TYPE (* logiBUS DI Events Struct Octal *)
  (* Version 1.0, 2026-05-28, franz *)
  PACKAGE logiBUS::io::DI;
  logiBUS_DI_Events_S_Octal : STRUCT
    Port1 : logiBUS::io::DI::logiBUS_DI_Events_S;
    Port2 : logiBUS::io::DI::logiBUS_DI_Events_S;
    Port3 : logiBUS::io::DI::logiBUS_DI_Events_S;
    Port4 : logiBUS::io::DI::logiBUS_DI_Events_S;
    Port5 : logiBUS::io::DI::logiBUS_DI_Events_S;
    Port6 : logiBUS::io::DI::logiBUS_DI_Events_S;
    Port7 : logiBUS::io::DI::logiBUS_DI_Events_S;
    Port8 : logiBUS::io::DI::logiBUS_DI_Events_S;
  END_STRUCT;
END_TYPE
